ABB RobotStudio station: Base1.rsstn

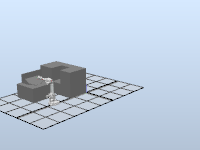
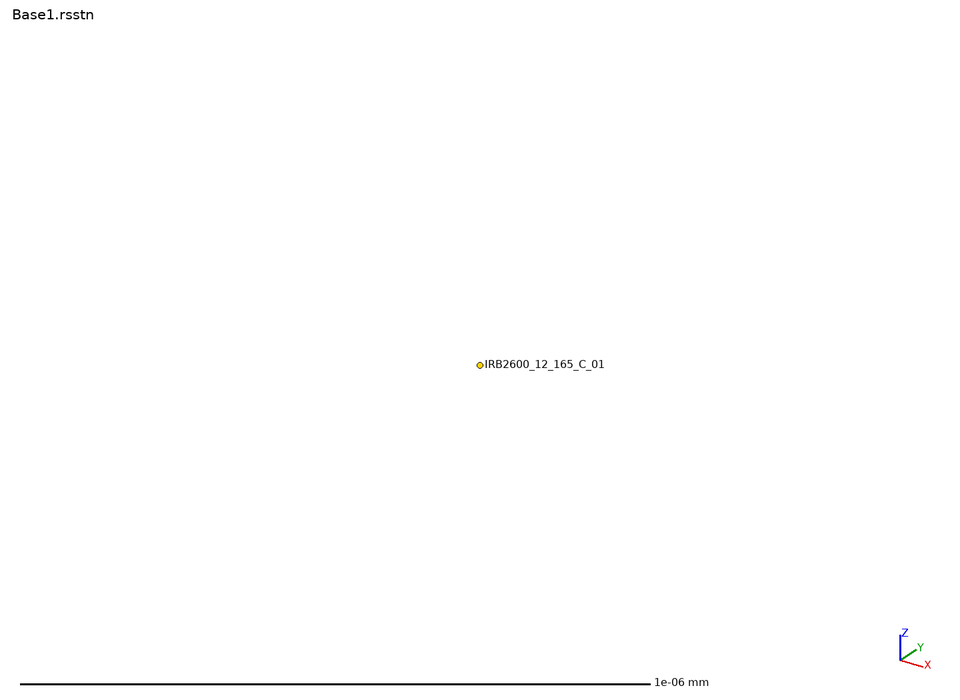
[picture v1: parts stored in the station drawn from their meshes, with robot base, taught points and paths (robot models come from the ABB library and are not in the file)]
Station Base1 (saved by RobotStudio 21.2.9526.0)
Controller Controlador4, task T_ROB1: task frame (RAPID world) sits at (0, 2644.78, 63.62) mm in the station
Controller Controlador4
  mechanical unit ROB_1: IRB2600_12_165_C_01, 6 joints, base frame (0, 0, 0) mm
Layout (positions relative to the parent item):
  - Torno_2 [part] at (0, 0, 1500) mm, size 2500 x 1300 x 1500 mm
  - Conjunto_para_piezas_3 [part] at (1054.46, 4084.49, 489.14) mm, rotated rx 90 ry 0 rz 0 deg, size 1400 x 1500 x 1500 mm
  - IRB2600_12_165_C_01 [mechanism] at (0, 2644.78, 63.62) mm; joint values [0.0804, 0.0165, -0.0774, -0.1254, 0.5896, -0.0887] (rad or m)
      links: Base, Link1, Link2, Link3, Link4, Link5, Link6
